// TIA Portal V16 export
// export: Created 2024-12-03T15:41:44.8646903Z, ExportSetting WithReadOnly, DisplayName Totally Integrated Automation Portal, DisplayVersion V16 Update 6, DisplayName TIA Portal Version Control Interface, DisplayVersion V16 Update 2, DisplayName TIA Portal Openness, DisplayVersion V16 Update 6, DisplayName TIA Portal Teamcenter Gateway, DisplayVersion V16, DisplayName SINAMICS Startdrive Advanced, DisplayVersion V16 Update 5, DisplayName SINAMICS Startdrive G130, G150, S120, S150, SINAMICS MV, S210, DisplayVersion V16 Update 5, DisplayName SINAMICS Startdrive G110M, G120, G120C, G120D, G120P, G115D, DisplayVersion V16 Update 5, DisplayName STEP 7 Professional, DisplayVersion V16 Update 6, DisplayName STEP 7 Safety, DisplayVersion V16, DisplayName WinCC Advanced / Unified PC, DisplayVersion V16 Update 6
TYPE "Motor_DOL_UDT"
// stored: CreationDate 2021-07-13T07:41:36.2278727Z, InterfaceModifiedDate 2020-12-13T14:34:57.5526505Z, IsConsistent true, LibraryConformanceStatus The object is library-conformant., ModifiedDate 2021-03-27T07:36:47.7019474Z
   STRUCT
      Cmd : Struct   // MotorCommands
         Reset : Bool;
         Interlock : Bool;
         OnAuto : Bool;
         OnManual : Bool;
         DirectionAuto : Bool;
         DirectionManual : Bool;
      END_STRUCT;
      Alarms : Struct
         NotOnTImedOut : "HmiAlarm";   // Motor not on in time
         NotOffTimedOut : "HmiAlarm";   // Motor not off in time
         ThermalProtection : "HmiAlarm";   // Motor thermal protection not ok
         AlarmStatus : Word;   // lsb 1 not on | lsb 2 not off | lsb 3 error from soft starter
      END_STRUCT;
      Status : Struct
         Interlocked : Bool;
         ManualModeActive : Bool;
         ManualCommandsDisabled : Bool;
         Running : Bool;
         Status : Word;   // lsb 0 interlocked | lsb 1 running | lbs2 manual mode active
      END_STRUCT;
      "Name" : String[20];
      Zone : Int := 1;
      Info { S7_SetPoint := 'True'} : "MotorInfo";
      CommonStatus : Int;
   END_STRUCT;
END_TYPE
